FUNCTION_BLOCK BtnRequestFBD
VAR_INPUT
	ixButtonElevat1 : BOOL ;
	ixButtonLevel1 : BOOL ;
	ixButtonElevat2 : BOOL ;
	ixButtonLevel2 : BOOL ;
	ixButtonElevat3 : BOOL ;
	ixButtonLevel3 : BOOL ;
END_VAR
VAR_OUTPUT
	ixQueue : BOOL ;
	iiQueueOrder : INT ;
END_VAR
VAR
END_VAR

IF ixButtonElevat1 OR ixButtonLevel1 THEN
	iiQueueOrder := 1 ;
	ixQueue := TRUE ;
ELSIF ixButtonElevat2 OR ixButtonLevel2 THEN
	iiQueueOrder := 2 ;
	ixQueue := TRUE ;
ELSIF ixButtonElevat3 OR ixButtonLevel3 THEN
	iiQueueOrder := 3 ;
	ixQueue := TRUE ;
ELSE
	iiQueueOrder := - 1 ;
	ixQueue := FALSE ;
END_IF

END_FUNCTION_BLOCK

(* stored: Version 1.1.0.1, ProductVersion 3.1.4024.12
   POU BtnRequestFBD: Id {b402b172-9920-48c7-ba62-269938338d0f}, SpecialFunc None *)
